TYPE ST_FeedbackLeica :
STRUCT
	pos: ARRAY[0..2] OF LREAL;
	R11: LREAL;
	R12: LREAL;
	R13: LREAL;
	R21: LREAL;
	R22: LREAL;
	R23: LREAL;
	R31: LREAL;
	R32: LREAL;
	R33: LREAL;
END_STRUCT
END_TYPE

(* stored: Version 1.1.0.1, ProductVersion 3.1.4026.8
   DUT ST_FeedbackLeica: Id {9230227a-713d-4e8d-a793-8a7c767d6582} *)
